PROGRAM ReadCSV
VAR
		
	sFileName		:STRING:='C:\TempSample\TextModeGen.csv';
	
	fbFileOpen: FB_FileOpen;
	//fbFilePuts: FB_FilePuts;
	fbFileGets: FB_FileGets;
	fbFileClose: FB_FileClose;
	bRead			:BOOL;
	iStep			:E_ReadCSVStep;
END_VAR

CASE iStep OF
	E_ReadCSVStep.Step_Init:
	
		IF	bRead THEN 
			bRead := FALSE;			
			iStep:=	E_ReadCSVStep.Step_Open;			
		END_IF
		
	E_ReadCSVStep.Step_Open: (*open source file*)
		fbFileOpen(sNetId:= ,sPathName:= ,nMode:= ,ePath:= ,bExecute:=FALSE,
					tTimeout:=T#3S ,bBusy=> ,bError=> ,nErrId=> ,hFile=> );
					
		fbFileOpen(sNetId:= ,sPathName:= sFileName,nMode:= FOPEN_MODEREAD OR FOPEN_MODETEXT  ,ePath:=PATH_GENERIC ,bExecute:=TRUE,
					tTimeout:=T#3S ,bBusy=> ,bError=> ,nErrId=> ,hFile=> );
		
		iStep := E_ReadCSVStep.Step_OpenWaite;
		
	E_ReadCSVStep.Step_OpenWaite:
		fbFileOpen(bExecute:=FALSE);
		IF NOT fbFileOpen.bBusy THEN 
			IF NOT fbFileOpen.bError THEN 
				iStep := E_ReadCSVStep.Step_ReadSingleLine;
			ELSE	(*error file not found?*)
				iStep := 
			END_IF			
		END_IF

	
END_CASE

END_PROGRAM

(* stored: Version 1.1.0.1, ProductVersion 3.1.4022.16
   POU ReadCSV: Id {8e1b1dca-04d3-4b70-90db-da206145f0ac}, SpecialFunc None *)
